Staubli VAL3: velOverwrite.pgx

public program velOverwrite(bool x_bOverwriteVel)
begin

  // Do nothing
  // See start() program for more details

end
